(* IEC 61131-3 sources: lpmlv2022/src/blocks/configurationBlocks, 5 files *)

(* ---- LPMLV2022_ConfigureCompleteCmdCfg.st ---- *)
NAMESPACE Simatic.Ax.LPMLV2022
///================================================================================
/// SIEMENS AG
/// (c)Copyright 2025 All Rights Reserved
///--------------------------------------------------------------------------------
/// Library: LPMLV2022
/// Engineering: SIMATIC AX
/// Restrictions: -
/// Requirements: S7-1500 FW 2.6
/// Functionality: The function generates a DWord value which represents
///                the state configuration for all unit modes.
///
///                Note: All inputs must be set to comply with ANSI/ISA-TR88.00.02-2022
///================================================================================
FUNCTION ConfigureCompleteCmdCfg
    VAR_INPUT
        /// TRUE: The Complete control command is taken into account in state Suspended
        Suspended : BOOL;
        /// TRUE: The Complete control command is taken into account in state Execute
        Execute : BOOL;
        /// TRUE: The Complete control command is taken into account in state Held
        Held : BOOL;
    END_VAR

    VAR_OUTPUT
        /// Complete control command configuration for all unit modes for direct connection
        /// with the input config.completeCmdCfg of the desired UnitModeStateManager instance.
        completeCmdCfg : DWORD;
    END_VAR

    // Initialize states configuration
    completeCmdCfg := DWORD#16#0000_0000;

    // Set states configuration
    completeCmdCfg.%X5 := Suspended;
    completeCmdCfg.%X6 := Execute;
    completeCmdCfg.%X11 := Held;

END_FUNCTION

END_NAMESPACE

(* ---- LPMLV2022_ConfigureDisabledStatesCfg.st ---- *)
NAMESPACE Simatic.Ax.LPMLV2022
///================================================================================
/// SIEMENS AG
/// (c)Copyright 2025 All Rights Reserved
///--------------------------------------------------------------------------------
/// Library: LPMLV2022
/// Engineering: SIMATIC AX
/// Restrictions: -
/// Requirements: S7-1500 FW 2.6
/// Functionality: The function generates a DWord value which represents
///                the state configuration for one unit mode.
///================================================================================
FUNCTION ConfigureDisabledStatesCfg
    VAR_INPUT
        /// TRUE: Disable state Clearing
        Clearing : BOOL;
        /// TRUE: Disable state Starting
        Starting : BOOL;
        /// TRUE: Disable state Suspended
        Suspended : BOOL;
        /// TRUE: Disable state Stopping
        Stopping : BOOL;
        /// TRUE: Disable state Aborting
        Aborting : BOOL;
        /// TRUE: Disable state Holding
        Holding : BOOL;
        /// TRUE: Disable state Held
        Held : BOOL;
        /// TRUE: Disable state Unholding
        Unholding : BOOL;
        /// TRUE: Disable state Suspending
        Suspending : BOOL;
        /// TRUE: Disable state Unsuspending
        Unsuspending : BOOL;
        /// TRUE: Disable state Resetting
        Resetting : BOOL;
        /// TRUE: Disable state Completing
        Completing : BOOL;
        /// TRUE: Disable state Completed
        Completed : BOOL;
    END_VAR

    VAR_OUTPUT
        /// Disabled states configuration for one unit mode for direct connection with the input
        /// config.DisabledStatesCfg[<unit mode>] of the desired UnitModeStateManager instance.
        DisabledStatesCfg : DWORD;
    END_VAR

    // Initialize states configuration
    DisabledStatesCfg := DWORD#16#0000_0000;

    // Note: Stopped (.%X2), Idle (.%X4), Execute (.%X6) and Aborted (.%X9) are always present. They cannot be disabled

    // Set states configuration
    DisabledStatesCfg.%X1 := Clearing;
    DisabledStatesCfg.%X3 := Starting;
    DisabledStatesCfg.%X5 := Suspended;
    DisabledStatesCfg.%X7 := Stopping;
    DisabledStatesCfg.%X8 := Aborting;
    DisabledStatesCfg.%X10 := Holding;
    DisabledStatesCfg.%X11 := Held;
    DisabledStatesCfg.%X12 := Unholding;
    DisabledStatesCfg.%X13 := Suspending;
    DisabledStatesCfg.%X14 := Unsuspending;
    DisabledStatesCfg.%X15 := Resetting;
    DisabledStatesCfg.%X16 := Completing;
    DisabledStatesCfg.%X17 := Completed;

END_FUNCTION

END_NAMESPACE

(* ---- LPMLV2022_ConfigureEnabledModesCfg.st ---- *)
NAMESPACE Simatic.Ax.LPMLV2022
///================================================================================
/// SIEMENS AG
/// (c)Copyright 2025 All Rights Reserved
///--------------------------------------------------------------------------------
/// Library: LPMLV2022
/// Engineering: SIMATIC AX
/// Restrictions: -
/// Requirements: S7-1500 FW 2.6
/// Functionality: The function generates the unit mode configuration as DWord.
///================================================================================
FUNCTION ConfigureEnabledModesCfg
    VAR_INPUT
        /// TRUE: Enable unit mode Production
        ProductionMode : BOOL;
        /// TRUE: Enable unit mode Maintenance
        MaintenanceMode : BOOL;
        /// TRUE: Enable user-defined unit mode 01
        UserMode01 : BOOL;
        /// TRUE: Enable user-defined unit mode 02
        UserMode02 : BOOL;
        /// TRUE: Enable user-defined unit mode 03
        UserMode03 : BOOL;
        /// TRUE: Enable user-defined unit mode 04
        UserMode04 : BOOL;
        /// TRUE: Enable user-defined unit mode 05
        UserMode05 : BOOL;
        /// TRUE: Enable user-defined unit mode 06
        UserMode06 : BOOL;
        /// TRUE: Enable user-defined unit mode 07
        UserMode07 : BOOL;
        /// TRUE: Enable user-defined unit mode 08
        UserMode08 : BOOL;
        /// TRUE: Enable user-defined unit mode 09
        UserMode09 : BOOL;
        /// TRUE: Enable user-defined unit mode 10
        UserMode10 : BOOL;
        /// TRUE: Enable user-defined unit mode 11
        UserMode11 : BOOL;
        /// TRUE: Enable user-defined unit mode 12
        UserMode12 : BOOL;
        /// TRUE: Enable user-defined unit mode 13
        UserMode13 : BOOL;
        /// TRUE: Enable user-defined unit mode 14
        UserMode14 : BOOL;
        /// TRUE: Enable user-defined unit mode 15
        UserMode15 : BOOL;
        /// TRUE: Enable user-defined unit mode 16
        UserMode16 : BOOL;
        /// TRUE: Enable user-defined unit mode 17
        UserMode17 : BOOL;
        /// TRUE: Enable user-defined unit mode 18
        UserMode18 : BOOL;
        /// TRUE: Enable user-defined unit mode 19
        UserMode19 : BOOL;
        /// TRUE: Enable user-defined unit mode 20
        UserMode20 : BOOL;
        /// TRUE: Enable user-defined unit mode 21
        UserMode21 : BOOL;
        /// TRUE: Enable user-defined unit mode 22
        UserMode22 : BOOL;
        /// TRUE: Enable user-defined unit mode 23
        UserMode23 : BOOL;
        /// TRUE: Enable user-defined unit mode 24
        UserMode24 : BOOL;
        /// TRUE: Enable user-defined unit mode 25
        UserMode25 : BOOL;
        /// TRUE: Enable user-defined unit mode 26
        UserMode26 : BOOL;
        /// TRUE: Enable user-defined unit mode 27
        UserMode27 : BOOL;
        /// TRUE: Enable user-defined unit mode 28
        UserMode28 : BOOL;
    END_VAR

    VAR_OUTPUT
        /// Enabled unit modes configuration for direct connection with the input config.EnabledModesCfg
        /// of the desired UnitModeStateManager instance
        EnabledModesCfg : DWORD;
    END_VAR

    // Initialize unitMode configuration
    EnabledModesCfg := DWORD#16#0000_0008; // Note: mode Manual (EnabledModesCfg.%X3) is mandatory

    // Set unitMode configuration
    EnabledModesCfg.%X1 := ProductionMode;
    EnabledModesCfg.%X2 := MaintenanceMode;
    EnabledModesCfg.%X4 := UserMode01;
    EnabledModesCfg.%X5 := UserMode02;
    EnabledModesCfg.%X6 := UserMode03;
    EnabledModesCfg.%X7 := UserMode04;
    EnabledModesCfg.%X8 := UserMode05;
    EnabledModesCfg.%X9 := UserMode06;
    EnabledModesCfg.%X10 := UserMode07;
    EnabledModesCfg.%X11 := UserMode08;
    EnabledModesCfg.%X12 := UserMode09;
    EnabledModesCfg.%X13 := UserMode10;
    EnabledModesCfg.%X14 := UserMode11;
    EnabledModesCfg.%X15 := UserMode12;
    EnabledModesCfg.%X16 := UserMode13;
    EnabledModesCfg.%X17 := UserMode14;
    EnabledModesCfg.%X18 := UserMode15;
    EnabledModesCfg.%X19 := UserMode16;
    EnabledModesCfg.%X20 := UserMode17;
    EnabledModesCfg.%X21 := UserMode18;
    EnabledModesCfg.%X22 := UserMode19;
    EnabledModesCfg.%X23 := UserMode20;
    EnabledModesCfg.%X24 := UserMode21;
    EnabledModesCfg.%X25 := UserMode22;
    EnabledModesCfg.%X26 := UserMode23;
    EnabledModesCfg.%X27 := UserMode24;
    EnabledModesCfg.%X28 := UserMode25;
    EnabledModesCfg.%X29 := UserMode26;
    EnabledModesCfg.%X30 := UserMode27;
    EnabledModesCfg.%X31 := UserMode28;

END_FUNCTION

END_NAMESPACE

(* ---- LPMLV2022_ConfigureHoldCmdCfg.st ---- *)
NAMESPACE Simatic.Ax.LPMLV2022
///================================================================================
/// SIEMENS AG
/// (c)Copyright 2025 All Rights Reserved
///--------------------------------------------------------------------------------
/// Library: LPMLV2022
/// Engineering: SIMATIC AX
/// Restrictions: -
/// Requirements: S7-1500 FW 2.6
/// Functionality: The function generates a DWord value which represents
///                the state configuration for all unit modes.
///
///                Note: Only the inputs 'Suspended' and 'Execute' must be set
///                      to comply with ANSI/ISA-TR88.00.02-2022
///================================================================================
FUNCTION ConfigureHoldCmdCfg
    VAR_INPUT
        /// TRUE: The Hold control command is taken into account in state Starting
        Starting : BOOL;
        /// TRUE: The Hold control command is taken into account in state Idle
        Idle : BOOL;
        /// TRUE: The Hold control command is taken into account in state Suspended
        Suspended : BOOL;
        /// TRUE: The Hold control command is taken into account in state Execute
        Execute : BOOL;
        /// TRUE: The Hold control command is taken into account in state Unholding
        Unholding : BOOL;
        /// TRUE: The Hold control command is taken into account in state Suspending
        Suspending : BOOL;
        /// TRUE: The Hold control command is taken into account in state Unsuspending
        Unsuspending : BOOL;
        /// TRUE: The Hold control command is taken into account in state Completing
        Completing : BOOL;
        /// TRUE: The Hold control command is taken into account in state Completed
        Completed : BOOL;
    END_VAR

    VAR_OUTPUT
        /// Hold control command configuration for all unit modes for direct connection
        /// with the input config.holdCmdCfg of the desired UnitModeStateManager instance
        holdCmdCfg : DWORD;
    END_VAR

    // Initialize states configuration
    holdCmdCfg := DWORD#16#0000_0000;

    // Set states configuration
    holdCmdCfg.%X3 := Starting;
    holdCmdCfg.%X4 := Idle;
    holdCmdCfg.%X5 := Suspended;
    holdCmdCfg.%X6 := Execute;
    holdCmdCfg.%X12 := Unholding;
    holdCmdCfg.%X13 := Suspending;
    holdCmdCfg.%X14 := Unsuspending;
    holdCmdCfg.%X16 := Completing;
    holdCmdCfg.%X17 := Completed;

END_FUNCTION

END_NAMESPACE

(* ---- LPMLV2022_ConfigureModeTransitionCfg.st ---- *)
NAMESPACE Simatic.Ax.LPMLV2022
///================================================================================
/// SIEMENS AG
/// (c)Copyright 2025 All Rights Reserved
///--------------------------------------------------------------------------------
/// Library: LPMLV2022
/// Engineering: SIMATIC AX
/// Restrictions: -
/// Requirements: S7-1500 FW 2.6
/// Functionality: The function generates a DWord value which represents
///                the state configuration for one unit mode.
///================================================================================
FUNCTION ConfigureModeTransitionCfg
    VAR_INPUT
        /// TRUE: Allow a mode transition to/from state Clearing
        Clearing : BOOL;
        /// TRUE: Allow a mode transition to/from state Stopped
        Stopped : BOOL;
        /// TRUE: Allow a mode transition to/from state Starting
        Starting : BOOL;
        /// TRUE: Allow a mode transition to/from state Idle
        Idle : BOOL;
        /// TRUE: Allow a mode transition to/from state Suspended
        Suspended : BOOL;
        /// TRUE: Allow a mode transition to/from state Execute
        Execute : BOOL;
        /// TRUE: Allow a mode transition to/from state Stopping
        Stopping : BOOL;
        /// TRUE: Allow a mode transition to/from state Aborting
        Aborting : BOOL;
        /// TRUE: Allow a mode transition to/from state Aborted
        Aborted : BOOL;
        /// TRUE: Allow a mode transition to/from state Holding
        Holding : BOOL;
        /// TRUE: Allow a mode transition to/from state Held
        Held : BOOL;
        /// TRUE: Allow a mode transition to/from state Unholding
        Unholding : BOOL;
        /// TRUE: Allow a mode transition to/from state Suspending
        Suspending : BOOL;
        /// TRUE: Allow a mode transition to/from state Unsuspending
        Unsuspending : BOOL;
        /// TRUE: Allow a mode transition to/from state Resetting
        Resetting : BOOL;
        /// TRUE: Allow a mode transition to/from state Completing
        Completing : BOOL;
        /// TRUE: Allow a mode transition to/from state Completed
        Completed : BOOL;
    END_VAR

    VAR_OUTPUT
        /// Mode Transition Configuration for one unit mode for direct connection with the input
        /// config.ModeTransitionCfg[<unit mode>] of the desired UnitModeStateManager instance
        ModeTransitionCfg : DWORD;
    END_VAR

    // Initialize states configuration
    ModeTransitionCfg := DWORD#16#0000_0000;

    // Set states configuration
    ModeTransitionCfg.%X1 := Clearing;
    ModeTransitionCfg.%X2 := Stopped;
    ModeTransitionCfg.%X3 := Starting;
    ModeTransitionCfg.%X4 := Idle;
    ModeTransitionCfg.%X5 := Suspended;
    ModeTransitionCfg.%X6 := Execute;
    ModeTransitionCfg.%X7 := Stopping;
    ModeTransitionCfg.%X8 := Aborting;
    ModeTransitionCfg.%X9 := Aborted;
    ModeTransitionCfg.%X10 := Holding;
    ModeTransitionCfg.%X11 := Held;
    ModeTransitionCfg.%X12 := Unholding;
    ModeTransitionCfg.%X13 := Suspending;
    ModeTransitionCfg.%X14 := Unsuspending;
    ModeTransitionCfg.%X15 := Resetting;
    ModeTransitionCfg.%X16 := Completing;
    ModeTransitionCfg.%X17 := Completed;

END_FUNCTION

END_NAMESPACE
